TYPE "Type_Motor"
VERSION : 0.1
   STRUCT
      timeout : Int;
      seq : Bool;
      opt : Bool;
      default : Bool;
      timeout2 : Int;
      typ : Int;   // tipo motore per nome e icona HMI
      diff : ULInt;
      diff2 : ULInt;
      seqok : Bool;
      timeoutbtn : Int;
      timeout3 : Int;
      timeout4 : Int;
   END_STRUCT;

END_TYPE

Class Motor(